Fanuc KAREL source: kc00008.KL

-- PROVISIONAL review KL for V1013-1; original PC SHA256 41e7721378a33654f0a2db3e1c7cefbcc8d578563b40d9833d76f2cb9734cde5
-- Incomplete behavior may be omitted. Consult companion uncertainty JSON. Do not deploy.
PROGRAM KC00008
%NOLOCKGROUP
BEGIN
  -- UNRESOLVED_PC offsets 5-33; opcodes 27,22,1C,22,22,31
  -- UNRESOLVED_PC offsets 38-42; opcodes 7F
END KC00008
